FUNCTION isOpen : BOOL
VAR_INPUT
	sensorID			:	DWORD;
END_VAR
VAR
	fbRecGeneric		: 	FB_Rec_Generic;
END_VAR

fbRecGeneric(str_KL6581 := GVL_EnOcean.stKL6581, byNode := 0, dw_ID := sensorID);

IF fbRecGeneric.ar_Value[3] = 8 THEN
	isOpen := TRUE;
ELSE
	isOpen := FALSE;
END_IF

END_FUNCTION

(* stored: Version 1.1.0.1, ProductVersion 3.1.4024.2
   POU isOpen: Id {48a17815-3d01-4dd8-9f86-4d30e0d44ec4}, SpecialFunc None *)
